TYPE ST_StorageStatus :
STRUCT
END_STRUCT
END_TYPE

(* stored: Version 1.1.0.1, ProductVersion 3.1.4024.13
   DUT ST_StorageStatus: Id {8b15e55f-e684-4d28-91a5-e9116232e5d3} *)
